PROGRAM ActuationSystems
VAR
fbMainJibCylinderHyd : ValveControlledCylinder;
fbKnuckleJibCylinderHyd : ValveControlledCylinder;
fbKingRotationCylinderHyd : ValveControlledCylinder;
//HydraulicCylinder
fbMainJibCylinderMech : CylinderMech;
fbKnuckleJibCylinderMech : CylinderMech;
fbkingRotationCylinderMech : CylinderMech;

fbFWKinematics : FWKinematics;
fbHPU : HPU;
END_VAR

fbHPU(
);

fbFWKinematics(
	L1 := 4.543126+1.097+1.000,  												//[m]
	L2 := 0,																	//[m]
	L3 := 17.939373,															//[m]
	L4 := 9.548784,																//[m]
	thetaMainBoom := ActuationSystems.fbKnuckleJibCylinderHyd.AngleJoint,		//[rad]
	thetaKnuckleBoom := ActuationSystems.fbMainJibCylinderHyd.AngleJoint, 		//[rad]
	thetaSlew := 0																//[rad]
);

//Hyd Model for MainJibCylinder
fbMainJibCylinderHyd(
	uDcvEnable := Inputs.uDcvEnableMainJib,
	uDcv := Inputs.uDcvMainJib,	
	ReturnPressure := G_ActuationSystems.ReturnPressure,
	SupplyPressure := G_ActuationSystems.SupplyPressure,
	par := Param.pMainJibCylinder,
	xPiston := fbMainJibCylinderMech.PistonPosition,
	vPiston := fbMainJibCylinderMech.PistonVelocity,
);
//Hyd Model for KnuckleJibCylinder
fbKnuckleJibCylinderHyd(
	uDcvEnable := Inputs.uDcvEnableKnuckleJib,
	uDcv := Inputs.uDcvKnuckleJib,	
	ReturnPressure := G_ActuationSystems.ReturnPressure,
	SupplyPressure := G_ActuationSystems.SupplyPressure,
	par := Param.pKnuckleJibCylinder,
	xPiston := fbKnuckleJibCylinderMech.PistonPosition,
	vPiston := fbKnuckleJibCylinderMech.PistonVelocity,
);
//Hyd Model for KingRotationCylinder
fbKingRotationCylinderHyd(
	uDcvEnable := Inputs.uDcvEnableKingRotation,
	uDcv := Inputs.uDcvKingRotation,	
	ReturnPressure := G_ActuationSystems.ReturnPressure,
	SupplyPressure := G_ActuationSystems.SupplyPressure,
	par := Param.pMainJibCylinder,
	xPiston := fbkingRotationCylinderMech.PistonPosition,
	vPiston := fbkingRotationCylinderMech.PistonVelocity,
);


//Temp Mechanical Model for MainJibCylinder
fbMainJibCylinderMech(
	F_Hydraulic := fbMainJibCylinderHyd.F_Hydraulic,
	param := Param.pMainJibCylinder,
	F_Piston => Work.FpistonMainJib
);	
//Temp Mechanical Model for KnuckleJibCylinder
fbKnuckleJibCylinderMech(
	F_Hydraulic := fbKnuckleJibCylinderHyd.F_Hydraulic,
	param := Param.pKnuckleJibCylinder,
	F_Piston => Work.FpistonKnuckleJib
);	
//Temp Mechanical Model for KingRotationCylinder
fbkingRotationCylinderMech(
	F_Hydraulic := fbKingRotationCylinderHyd.F_Hydraulic,
	param := Param.pKingRotationCylinder,
	F_Piston => Work.FpistonKingRotation
);

END_PROGRAM

(* stored: Version 1.1.0.1, ProductVersion 3.1.4024.9
   POU ActuationSystems: Id {3cabdd9c-217f-443b-9923-404fabc5dbf5}, SpecialFunc None *)
